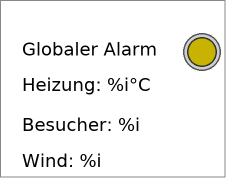
VISUALIZATION Zentrale  // 226x178
    Lamp1 (180,30 44x44), variable: net_einbruch_alarm, style: Lamp-Lamp1-Yellow
    Label (19,35 191x29), "Globaler Alarm"
    Textfield (19,70 150x30), "Heizung: %i°C", text variable: net_heizung_out
    Textfield (19,110 150x30), "Besucher: %i", text variable: GL_Besucher
    Textfield (19,146 150x30), "Wind: %i", text variable: net_wind
END_VISUALIZATION

(* stored: Version 1.1.0.1, ProductVersion 3.1.4018.5
   Visu Zentrale: Id {146fe0b1-258a-442b-9821-1b243a9cf5ea} *)
